PROGRAM P3_00_MAIN
VAR
	tonDeleteDelay			:TON;
END_VAR

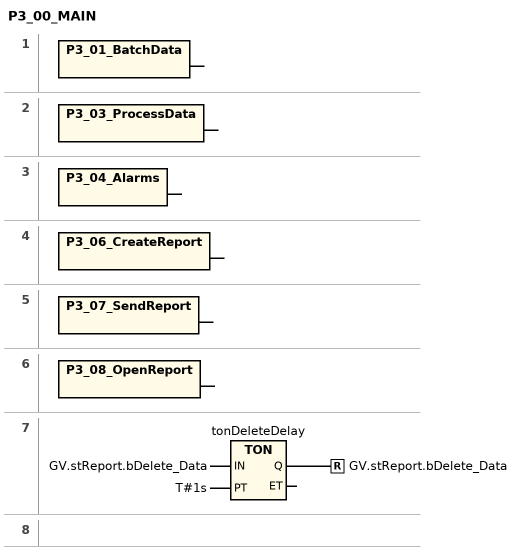
// NETWORK 1
P3_01_BatchData();

// NETWORK 2
P3_03_ProcessData();

// NETWORK 3
P3_04_Alarms();

// NETWORK 4
P3_06_CreateReport();

// NETWORK 5
P3_07_SendReport();

// NETWORK 6
P3_08_OpenReport();

// NETWORK 7
tonDeleteDelay(IN := GV.stReport.bDelete_Data, PT := T#1s); // TON
GV.stReport.bDelete_Data R= tonDeleteDelay.Q;

// NETWORK 8

END_PROGRAM

(* stored: Version 1.1.0.1
   POU P3_00_MAIN: Id {6dbcf589-6ccb-47fd-98a1-d1c85a02152b}, SpecialFunc None *)
